    |   global total_dis = wv_total_hz * wave_dis
    | 
    |   # robot speed distance/time = speed
    |   wv_system_speed = total_dis / (wv_times)
    |   if(wv_times == 0 or cir_speed_org == 0):
    |     write_port_register(142,111)
    |     sleep(0.5)
    |     halt
    |   end
    |   return wv_system_speed
    | end
    | 
    | 
    | def set_current_voltage(o_cur,o_vol):
    |   if(isHicomm):
    |     set_current_voltage_hicomm(o_cur,o_vol)
    |   else:
    |     set_current_voltage_analog(o_cur,o_vol)
    |   end
    | end
    | 
    | def set_current_voltage_hicomm(o_cur,o_vol):
    |     write_port_register(204,o_cur)
    |     write_port_register(205,o_vol*10)
    |     write_port_register(133,o_cur)
    |     write_port_register(134,o_vol*10)
    | end
    | 
    | def set_current_voltage_analog(o_cur,o_vol):
    |     vol_an=((o_vol-14)/2.8)/10
    |     amp_an=((o_cur-60)/44)/10
    |     set_standard_analog_out(0,vol_an)
    |     set_standard_analog_out(1,amp_an)
    |     write_port_register(133,o_cur)
    |     write_port_register(134,o_vol*10)
    | end
    | 
    | def calculate_2f(wving_amplitude,tg_wv_wp1,tg_wv_wp2,cir_speed_org,wving_frequency,wving_delay,wving_crater,wving_dir):
    |   # 진폭
    |   global y_radius = wving_amplitude / 2
    |   # 이동 거리
    |   global move_dis = point_dist(tg_wv_wp1,tg_wv_wp2)*1000
    |   global move_dis_total = move_dis
    |   # total running time (sec) - cir_speed_org cpm.
    |   global wv_times_org = move_dis/(cir_speed_org/6)
    |   global wv_times = wv_times_org
    |   global wv_total_hz = floor(wv_times_org*wving_frequency/(1+wving_delay[0]+wving_delay[1]+wving_delay[2]+wving_delay[3]))
    |   global get_total = wv_total_hz
    | 
    |   dir=1
    | 
    |   ratio_t_sam = 1/get_total
    |   T1_sam = interpolate_pose(tg_wv_wp1,tg_wv_wp2,ratio_t_sam)
    |   ratio_t_sam = ratio_t_sam + 1/get_total
    |   T2_sam = interpolate_pose(tg_wv_wp1,tg_wv_wp2,ratio_t_sam)
    |   ratio_t_sam = ratio_t_sam + 1/get_total
    |   T3_sam = interpolate_pose(tg_wv_wp1,tg_wv_wp2,ratio_t_sam)
    | 
    |   push_angle = wving_crater[6]
    |   push_dis_sam = norm(y_radius)/tan(d2r(push_angle))
    |   Tp1_sam = feature_offset(T2_sam,p[0,y_radius/1000,0,0,0,0],wv_Line_Feature2)
    |   Tp2_sam = feature_offset(T2_sam,p[0,-y_radius/1000,0,0,0,0],wv_Line_Feature2)
    |   Tp1_sam = feature_offset(Tp1_sam,p[wving_dir*push_dis_sam/1000,0,0,0,0,0],wv_Line_Feature2)
    |   Tp3_sam = feature_offset(T3_sam,p[0,-y_radius/1000,0,0,0,0],wv_Line_Feature2)
    |   total_step = (get_line_dist(Tp1_sam,Tp2_sam)+get_line_dist(Tp1_sam,Tp3_sam))*1000
    |   total_dis = wv_total_hz * total_step
    | 
    |   wv_system_speed = (total_dis / wv_times)
    | 
    |   if(wv_times == 0 or cir_speed_org == 0):
    |     write_port_register(142,111)
    |     sleep(0.5)
    |     halt
    |   end
    |   return wv_system_speed
    | end
    | def weaving_simple(wv_wp1,wv_wp3,cir_speed_org,wving_frequency,wving_amplitude,welding_on):
    |   wv_dist = 0
    |   tilt_deg = [0,0,0]
    |   wving_delay = [0,0,0,0]
    |   wving_type = 1
    |   Arc_sen=[0,0,0,0,0,0]
    |   wv_gap=[0,0,0,0]
    |   welding_dir=1
    |   z_param=[0,0,0,0,0]
    |   par_2f=False
    |   wving_crater=[0,0,0,0,0,0,0,0,0,0]
    |   ext_fun=[0,0,0,0,0,0,0,0,0,0,0]
    |   wv_seq = [0,-1]
    |   wv_feature=p[0,0,0,0,0,0]
    |   wv_weldpar=[0,cir_speed_org,0,wving_frequency,wving_amplitude,wving_type,welding_dir]
    |   line_weaving_tp(wv_wp1,wv_wp3,wv_weldpar,tilt_deg,wving_delay,welding_on,Arc_sen,wv_gap,z_param,par_2f,wving_crater,ext_fun,wv_seq,wv_feature)
    | end
    | 
    | def line_weaving_tp(wv_wp1,wv_wp3,wv_weldpar=[100,10,0,1,5,1,1,1,0],tilt_deg=[0,0,0],wving_delay=[0,0,0,0],welding_on=False,Arc_sen=[0,0,0,0,0,0],wv_gap=[0,0,0,0],z_param=[0,0,0,0,0],par_2f=False,wving_crater=[0,0,0,0,0,0,0,0,0,0],ext_fun=[0,0,0,0,0,0,0,0,0,0,0],wv_seq = [0,-1],wv_feature=p[0,0,0,0,0,0]):
    |   global start_gas_time = 2
    |   global counter_average = 1
    |   global counter_average_num = 0
    |   global waste_cycle = ext_fun[8]
    |   if(first_half):
    |     Arc_sen[1] = Arc_sen[1]/2
    |     Arc_sen[2] = Arc_sen[2]/2
    |     Arc_sen[3] = Arc_sen[3]/2
    |     Arc_sen[4] = Arc_sen[4]/2
    |   end
    |   global arc_x_off=0
    |   global arc_z_off=0
    |   global Up = 0
    |   global Ui = 0
    |   global Up_z = 0
    |   global Ui_z = 0
    |   if(wv_weldpar[7] == 1):
    |     global record_multi = False
    |   else:
    |     global record_multi = True
    |   end
    |   global th_ext_fun = ext_fun
    |   RTDE_init()
    | 
    |   # e-Series 2, CB-Seris 8
    |   global system_bus_ms = 2
    | 
    |   global sin_dir = wv_seq[1]
    |   global start_trig = False
    |   dir=1
    |   if(par_2f):
    |     global squash_cycle = 0
    |     # sin_dir = sin_dir
    |     sin_dir = sin_dir * -1
    |   else:
    |     global squash_cycle = ext_fun[7]
    |   end
    |   global tri_count=0
    | 
    |   global z_bottom = z_param[0]/1000
    |   if(wv_weldpar[6]==-1):
    |     #right
    |     global vir_v = -1
    |   else:
    |     #left
    |     global vir_v = 1
    |   end
    | 
    |   if(par_2f):
    |     global cal_off_ang_rx = 1
    |     global cal_off_ang_ry = 0
    |   else:
    |     global cal_off_ang_rx = 0
    |     global cal_off_ang_ry = 1
    |   end
    | 
    |   if(wv_seq[0] == 2 or wv_seq[0] == 3):
    |     tilt_deg = [0,0,0]
    |     global cal_off_ang_rx = 0
    |     global cal_off_ang_ry = 0
    |   end
    | 
    |   global wv_Line_Feature2 = wv_wp1
    |   if(wv_weldpar[0] > 650 and par_2f == False):
    |     wv_weldpar[0] = 650
    |   end
    |   if(wv_wp3==p[0,0,0,0,0,0]):
    |     global wv_wp2 = feature_offset(wv_wp1,p[wv_weldpar[0]/1000,0,0,0,0,0],wv_Line_Feature2)
    |   else:
    |     global wv_wp2 = wv_wp3
    |     wv_weldpar[0] = point_dist(wv_wp1,wv_wp2)*1000
    |     global wv_dist_bak = point_dist(wv_wp1,wv_wp2)*1000
    |   end
    |   if(wv_feature != p[0,0,0,0,0,0]):
    |     wv_Line_Feature2 = wv_feature
    |   end
    |   if(vir_v==1):
    |     line_x = get_feature_Line(wv_wp1,wv_wp2)
    |   else:
    |     line_x = get_feature_Line(wv_wp2,wv_wp1)
    |   end
    |   pp1 = feature_offset(wv_wp1,p[0,20/1000,0,0,0,0],line_x)
    |   pp2 = pose_add(wv_wp1,p[0,0,20/1000,0,0,0])
    |   global wp_Feature = get_feature_plane_yz(wv_wp1,pp1,pp2)
    | 
    |   #setting
    |   if(par_2f):
    |     #todo - 1
    |     global offset_2f_k = -1 * ext_fun[9]
    |     global offset_2f_z = 1 * ext_fun[10]
    |     if(wv_seq[0] == 0 or wv_seq[0] == 1):
    |       # line_feature = get_feature_Line(wv_wp1,wv_wp2)
    |       line_feature = get_feature_Line(wv_wp2,wv_wp1)
    |       b_p1 = wv_wp1
    |       b_p2 = feature_offset(wv_wp1,p[0,0.02*vir_v,0,0,0,0],line_feature)
    |       # b_p2 = feature_offset(wv_wp1,p[0,0.01,0,0,0,0],line_feature)
    |       b_p3 = pose_add(wv_wp1,p[0,0,0.02,0,0,0])
    | 
    |       global back_feature = get_feature_plane_xz(b_p1,b_p2,b_p3)
    | 
    |       wv_wp1 = pose_trans(wv_wp1,p[0,0,0,0,0,d2r(-90)])
    |       wv_wp1 = feature_offset(wv_wp1,p[0,offset_2f_k/1000,0,0,0,0],back_feature)
    |       wv_wp1 = pose_add(wv_wp1,p[0,0,offset_2f_z/1000,0,0,0])
    |       global bak_wv_wp1 = wv_wp1
    |     end
    |       wv_wp2 = feature_offset(wv_wp2,p[0,offset_2f_k/1000,0,0,0,0],back_feature)
    |       wv_wp2 = pose_add(wv_wp2,p[0,0,offset_2f_z/1000,0,0,0])
    |       wv_wp2 = p[wv_wp2[0],wv_wp2[1],wv_wp2[2],wv_wp1[3],wv_wp1[4],wv_wp1[5]]
    |       global bak_wv_wp2 = wv_wp2
    |   end
    |   if(ext_fun[2]==1 and par_2f==False):
    |     w_voltage = ext_fun[3]
    |     w_current = ext_fun[4]
    |     set_current_voltage(w_current,w_voltage)
    |     global cir_speed_org_bak = wv_weldpar[1]
    |     global wving_amplitude_bak = wv_weldpar[4]
    |     wv_weldpar[1] = ext_fun[6]
    |     wv_weldpar[4] = ext_fun[5]
    |   end
    |   if(par_2f):
    |     global wv_system_speed = calculate_2f(wv_weldpar[4],wv_wp1,wv_wp2,wv_weldpar[1],wv_weldpar[3],wving_delay,wving_crater,wv_weldpar[6])
    |   else:
    |     global wv_system_speed = calculate_3f(wv_weldpar[4],wv_wp1,wv_wp2,wv_weldpar[1],wv_weldpar[3],wving_delay)
    |     x_radius = x_radius / 1000
    |   end
    |   global wv_set_speed = wv_system_speed
    |   ratio_t=0
    |   global y_radius = y_radius / 1000
    |   global y_radius_bak = y_radius
    |   global ext_stick = 0
    |   global th_arc_sen=Arc_sen
    |   global th_wv_gap=wv_gap
    |   global th_tilt_deg=tilt_deg
    |   global last_tilt_deg = th_tilt_deg
    |   global last_wv_wp1 = wv_wp1
    |   global last_wv_line = wv_Line_Feature2
    |   global last_z_bottom = z_bottom
    |   global th_wving_crater=wving_crater
    |   global th_par_2f = par_2f
    |   global th_cir_speed_org=wv_weldpar[1]
    |   global th_wv_wp1 = wv_wp1
    |   global th_wv_wp2 = wv_wp2
    |   global th_wv_wp3 = wv_wp3
    |   global th_wv_weldpar=wv_weldpar
    |   global th_wving_delay=wving_delay
    |   global th_z_param=z_param
    |   global th_wv_seq = wv_seq
    |   global th_wv_feature=wv_feature
    |   global th_dir = dir
    | 
    |   # if want to use approach position
    |   if(wv_seq[0] ==0 or wv_seq[0] == 1):
    |     global get_angle_rx = welding_angle_cal_2f(wv_wp1[1],tilt_deg,vir_v,cal_off_ang_rx)
    |     global get_angle_ry = welding_angle_cal_3f(wv_wp1[2],tilt_deg,z_bottom,cal_off_ang_ry)
    | 
    |     target_p = feature_offset(wv_wp1,p[0,0,0,d2r(tilt_deg[0] + get_angle_rx),d2r(tilt_deg[1] + get_angle_ry),d2r(tilt_deg[2])],wv_Line_Feature2)
    | 
    |     if(wv_weldpar[2]==1):
    |       target_p_appr = feature_offset(target_p,p[0,0,-0.02,0,0,0],wv_Line_Feature2)
    |       movel(target_p_appr,a=0.5,v=0.125)
    |     end
    |     movel(target_p,a=0.5,v=0.125)
    |   end
    |   CThread = run CalThread()
    |   DThread = run diff_Thread()
    |   TThread = run thread_timer()
    |   AThread = run Arc_Thread()
    |   TTRRhread = run thread_dist_rec()
    | 
    |   global timer_counting=True
    |   global program_weld_on = True
    | 
    |   if(a9_wv_weldingon==True):
    |     while(welding_off_t==55):
    |       sync()
    |     end
    |     if(wving_crater[2]>0):
    |       set_current_voltage(wving_crater[0],wving_crater[1])
    |     end
    |     if(welding_off_t != 1):
    |       if(isHicomm):
    |         write_welder(0,True)
    |       else:
    |         set_standard_digital_out(0,True)
    |       end
    |       while(read_welder(5)==False):
    |         if(weld_onoff==False):
    |             write_welder(0,True)
    |         end
    |         sync()
    |       end
    |       if(wving_crater[2]>0):
    |         #Crater Begin option
    |         write_output_float_register(1,1)
    |         sleep(wving_crater[2])
    |         set_current_voltage(ext_fun[1],ext_fun[0])
    |       end
    |     end
    |   end
    |   start_gas_time = 0
    | 
    |   background_cal=1
    |   background_ready=0
    |   FT_trig=True
    |   timer_1_is_counting = True
    |   global welding_program = False
    | 
    |   while((ratio_t < 1)):
    |     if( (norm(tri_count)>=2 and par_2f==False or FT_trig==True) or (norm(tri_count)>=4 and par_2f or FT_trig==True) ):
    |       FT_trig = False
    |       while(background_ready==0):
    |         sync()
    |       end
    |       tri_count = 0
    |       background_ready = 0
    |       global move_p = background_pose
    |       wv_wp2 = th_wv_wp2
    |       if(par_2f):
    |         background_cal=1
    |       else:
    |         background_cal=1
    |       end
    |       global a_val = 3
    |       if(a_val >= 30):
    |         write_port_register(142,112)
    |         sleep(0.5)
    |         halt
    |       end
    |     end
    |     if(wv_weldpar[5] ==1):
    |         if( (sin_dir==1 and wving_delay[0]==0) or (sin_dir==-1 and wving_delay[2]==0)):
    |          tri_count = tri_count + 1
    |         end
    |         global target_p = move_p[tri_count]
    |         # write_output_float_register(24,tri_count)
    |         # target_p=p[target_p[0],target_p[1],target_p[2],target_p[3],target_p[4],target_p[5]]
    |         tri_count = tri_count + 1
    |     elif(wv_weldpar[5] ==2):
    |       if((tri_count==0 and wving_delay[2]==0) or (tri_count==2 and wving_delay[0]==0)):
    |        tri_count = tri_count + 1
    |       end
    |       global target_p = move_p[tri_count]
    |       # write_output_float_register(24,tri_count)
    |       # target_p=p[target_p[0],target_p[1],target_p[2],target_p[3],target_p[4],target_p[5]]
    |       tri_count = tri_count + 1
    |     else:
    |       popup("Please insert 0 - sin or 1 - triangle")
    |     end
    |     if(target_p == p[0,0,0,0,0,0]):
    |       target_p = get_actual_tcp_pose()
    |     end
    |     #3F tri_count 2 는 tri_count가 계속 move_p[1]만 간다
    | 
    |     # write_output_float_register(23,sin_dir)
    | 
    |     ARC_T_ONOFF = True
    |     ARC_T_s_pose = get_actual_tcp_pose()
    |     ARC_T_e_pose = target_p
    |     if((norm(tri_count)== 2) and wving_delay[1]>0 and par_2f):
    |       #down
    |       movel(target_p,a=a_val,v=wv_system_speed/1000)
    |       sleep(wving_delay[1])
    |     elif((norm(tri_count)== 4) and wving_delay[3]>0 and par_2f):
    |       #4
    |       movel(target_p,a=a_val,v=wv_system_speed/1000)
    |       sleep(wving_delay[3])
    |     elif((norm(tri_count)== 2) and sin_dir==1 and wving_delay[1]>0 and par_2f == False):
    |       movel(target_p,a=a_val,v=wv_system_speed/1000)
    |       sleep(wving_delay[1])
    |     elif((norm(tri_count)== 2) and sin_dir==-1 and wving_delay[3]>0 and par_2f == False):
    |       movel(target_p,a=a_val,v=wv_system_speed/1000)
    |       sleep(wving_delay[3])
    |     elif((norm(tri_count)== 1) and wving_delay[2]>0 and par_2f):
    |       movel(target_p,a=a_val,v=wv_system_speed/1000)
    |       sleep(wving_delay[2])
    |     elif((norm(tri_count)== 3) and wving_delay[0]>0 and par_2f):
    |       #3
    |       movel(target_p,a=a_val,v=wv_system_speed/1000)
    |       sleep(wving_delay[0])
    |     else:
    |       movel(target_p,a=a_val,v=wv_system_speed/1000)
    |     end
    |     global last_pose = target_p
    |   end
    |   timer_1_is_counting = False
    | 
    |   if(a9_wv_weldingon == True and wving_crater[5]!=0):
    |     #crater end option
    |     set_current_voltage(wving_crater[3],wving_crater[4])
    |     sleep(wving_crater[5])
    |     program_weld_on = False
    |     set_current_voltage(ext_fun[1],ext_fun[0])
    |     if(isHicomm):
    |       write_port_register(202,0)
    |       write_port_register(149,0)
    |     else:
    |       set_standard_digital_out(0,False)
    |     end
    |     while(read_welder(5)==True):
    |       if(weld_onoff==True):
    |         write_welder(0,False)
    |       end
    |       sync()
    |     end
    |   end
    |   timer_counter = 0
    |   kill CThread
    |   kill DThread
    |   kill TThread
    |   kill AThread
    |   kill TTRRhread
    |   ARC_T_ONOFF=False
    |   timer_counter = 0
    |   timer_counting = False
    |   wcr_counter = 0
    |   wcr_counting = False
    |   get_wcr = False
    |   welding_off_t = 0
    |   plus_alpha_x = 0
    |   plus_alpha_z = 0
    | 
    |   if(wv_seq[0] == 0 or wv_seq[0] == 3):
    |     if(a9_wv_weldingon==True):
    |       program_weld_on = False
    |       write_port_register(202,0)
    |       write_port_register(149,0)
    |       write_welder(0,False)
    |       if(wv_weldpar[2]==1):
    |         target_pos = feature_offset(get_actual_tcp_pose(),p[0,0,-0.01,0,0,0],wv_Line_Feature2)
    |         movel(target_pos,0.5,0.01)
    |       end
    |     end
    |   end
    |   background_pose = [dumy_p,dumy_p,dumy_p,dumy_p]
    |   move_p = background_pose
    |   return sin_dir
    | end
    | 
    | 
    | def line_weaving_tp_l(wv_wp1,wv_wp3,wv_weldpar=[100,10,0,1,5,1,1,1,0],tilt_deg=[0,0,0],wving_delay=[0,0,0,0],welding_on=False,Arc_sen=[0,0,0,0,0,0],wv_gap=[0,0,0,0],z_param=[0,0,0,0,0],par_2f=False,wving_crater=[0,0,0,0,0,0,0,0,0,0],ext_fun=[0,0,0,0,0,0,0,0,0,0,0],wv_seq = [0,-1],wv_feature=p[0,0,0,0,0,0]):
    |   global start_gas_time = 2
    |   global counter_average = 1
    |   global counter_average_num = 0
    |   global waste_cycle = ext_fun[8]
    |   if(first_half):
    |     Arc_sen[1] = Arc_sen[1]/2
    |     Arc_sen[2] = Arc_sen[2]/2
    |     Arc_sen[3] = Arc_sen[3]/2
    |     Arc_sen[4] = Arc_sen[4]/2
    |   end
    |   global current_list = 0
    |   global wv_wp4 = wv_wp3
    |   global A_T1 = wv_wp4[0]
    |   global A_T2 = wv_wp4[1]
    |   global A_T3 = wv_wp4[2]
    | 
    |   global arc_x_off=0
    |   global arc_z_off=0
    |   global Up = 0
    |   global Ui = 0
    |   global Up_z = 0
    |   global Ui_z = 0
    |   global th_ext_fun = ext_fun
    |   if(wv_weldpar[7] == 1):
    |     global record_multi = False
    |   else:
    |     global record_multi = True
    |   end
    |   RTDE_init()
    | 
    |   if (wv_gap[0]==1):
    |     gap_check = True
    |     wv_gap[0]=0
    |   else:
    |     gap_check= False
    |   end
    |   # e-Series 2, CB-Seris 8
    |   global system_bus_ms = 2
    | 
    |   global sin_dir = wv_seq[1]
    |   if(par_2f):
    |     global squash_cycle = 0
    |     # sin_dir = sin_dir
    |     sin_dir = sin_dir * -1
    |   else:
    |     global squash_cycle = ext_fun[7]
    |   end
    |   global start_trig = False
    |   dir=1
    | 
    |   global tri_count=0
    | 
    |   global z_bottom = z_param[0]/1000
    |   if(wv_weldpar[6]==-1):
    |     global vir_v = -1
    |   else:
    |     global vir_v = 1
    |   end
    | 
    |   if(par_2f):
    |     global cal_off_ang_rx = 1
    |     global cal_off_ang_ry = 0
    |   else:
    |     global cal_off_ang_rx = 0
    |     global cal_off_ang_ry = 1
    |   end
    | 
    |   if(wv_seq[0] == 2 or wv_seq[0] == 3):
    |     tilt_deg = [0,0,0]
    |     global cal_off_ang_rx = 0
    |     global cal_off_ang_ry = 0
    |   end
    | 
    |   global wv_Line_Feature2 = wv_wp1
    |   if(wv_weldpar[0] > 700 and par_2f == False):
    |     wv_weldpar[0] = 700
    |   end
    |   if(wv_wp3[0]==p[0,0,0,0,0,0]):
    |     global wv_wp2 = feature_offset(wv_wp1,p[wv_weldpar[0]/1000,0,0,0,0,0],wv_Line_Feature2)
    |   else:
    |     global wv_wp2 = wv_wp4[0]
    |     wv_weldpar[0] = point_dist(wv_wp1,wv_wp2)*1000
    |     global wv_dist_bak = point_dist(wv_wp1,wv_wp2)*1000
    |   end
    |   if(wv_seq[0] == 2 or wv_seq[0] == 3):
    |     wv_Line_Feature2 = wv_feature
    |   end
    |   if(vir_v==1):
    |     line_x = get_feature_Line(wv_wp1,wv_wp2)
    |   else:
    |     line_x = get_feature_Line(wv_wp2,wv_wp1)
    |   end  pp1 = feature_offset(wv_wp1,p[0,20/1000,0,0,0,0],line_x)
    |   pp2 = pose_add(wv_wp1,p[0,0,20/1000,0,0,0])
    |   global wp_Feature = get_feature_plane_yz(wv_wp1,pp1,pp2)
    | 
    |   #setting
    |   if(par_2f):
    |     #todo - 1
    |     offset_2f_k = -1 * ext_fun[9]
    |     offset_2f_z = 1 * ext_fun[10]
    |     if(wv_seq[0] == 0 or wv_seq[0] == 1):
    |       line_feature = get_feature_Line(wv_wp1,wv_wp2)
    |       b_p1 = wv_wp1
    |       b_p2 = feature_offset(wv_wp1,p[0,0.01*vir_v,0,0,0,0],line_feature)
    |       b_p3 = pose_add(wv_wp1,p[0,0,0.01,0,0,0])
    | 
    |       back_feature = get_feature_plane_xz(b_p1,b_p2,b_p3)
    |       wv_wp1 = pose_trans(wv_wp1,p[0,0,0,0,0,d2r(-90)])
    |       wv_wp1 = feature_offset(wv_wp1,p[0,offset_2f_k/1000,0,0,0,0],back_feature)
    |       wv_wp1 = pose_add(wv_wp1,p[0,0,offset_2f_z/1000,0,0,0])
    |       # wv_wp1 = pose_add(wv_wp1,p[offset_2f_k/1000,0,0,0,0,0])
    |     end
    |       # wv_wp2 = pose_add(wv_wp2,p[offset_2f_k/1000,0,0,0,0,0])
    |       wv_wp2 = feature_offset(wv_wp2,p[0,offset_2f_k/1000,0,0,0,0],back_feature)
    |       wv_wp2 = pose_add(wv_wp2,p[0,0,offset_2f_z/1000,0,0,0])
    |       wv_wp2 = p[wv_wp2[0],wv_wp2[1],wv_wp2[2],wv_wp1[3],wv_wp1[4],wv_wp1[5]]
    | 
    |       wv_wp3_p = feature_offset(wv_wp3[0],p[0,offset_2f_k/1000,0,0,0,0],back_feature)
    |       wv_wp3_p = pose_add(wv_wp3_p,p[0,0,offset_2f_z/1000,0,0,0])
    |       wv_wp3_p = p[wv_wp3_p[0],wv_wp3_p[1],wv_wp3_p[2],wv_wp1[3],wv_wp1[4],wv_wp1[5]]
    |       wv_wp4[0] = p[wv_wp3_p[0],wv_wp3_p[1],wv_wp3_p[2],wv_wp1[3],wv_wp1[4],wv_wp1[5]]
    | 
    |       wv_wp3_p = feature_offset(wv_wp3[1],p[0,offset_2f_k/1000,0,0,0,0],back_feature)
    |       wv_wp3_p = pose_add(wv_wp3_p,p[0,0,offset_2f_z/1000,0,0,0])
    |       wv_wp3_p = p[wv_wp3_p[0],wv_wp3_p[1],wv_wp3_p[2],wv_wp1[3],wv_wp1[4],wv_wp1[5]]
    |       wv_wp4[1] = p[wv_wp3_p[0],wv_wp3_p[1],wv_wp3_p[2],wv_wp1[3],wv_wp1[4],wv_wp1[5]]
    | 
    |       wv_wp3_p = feature_offset(wv_wp3[2],p[0,offset_2f_k/1000,0,0,0,0],back_feature)
    |       wv_wp3_p = pose_add(wv_wp3_p,p[0,0,offset_2f_z/1000,0,0,0])
    |       wv_wp3_p = p[wv_wp3_p[0],wv_wp3_p[1],wv_wp3_p[2],wv_wp1[3],wv_wp1[4],wv_wp1[5]]
    |       wv_wp4[2] = p[wv_wp3_p[0],wv_wp3_p[1],wv_wp3_p[2],wv_wp1[3],wv_wp1[4],wv_wp1[5]]
    |   end
    |   if(ext_fun[2]==1 and par_2f==False):
    |     #squash
    |     w_voltage = ext_fun[3]
    |     w_current = ext_fun[4]
    |     set_current_voltage(w_current,w_voltage)
    |     global cir_speed_org_bak = wv_weldpar[1]
    |     global wving_amplitude_bak = wv_weldpar[4]
    |     wv_weldpar[1] = ext_fun[6]
    |     wv_weldpar[4] = ext_fun[5]
    |   end
    |   if(par_2f):
    |     global wv_system_speed = calculate_2f(wv_weldpar[4],wv_wp1,wv_wp2,wv_weldpar[1],wv_weldpar[3],wving_delay,wving_crater,wv_weldpar[6])
    |   else:
    |     global wv_system_speed = calculate_3f(wv_weldpar[4],wv_wp1,wv_wp2,wv_weldpar[1],wv_weldpar[3],wving_delay)
    |     x_radius = x_radius / 1000
    |   end
    |   global wv_set_speed = wv_system_speed
    |   ratio_t=0
    |   # mm -> m
    |   global y_radius = y_radius / 1000
    |   global y_radius_bak = y_radius
    |   #init for thread
    |   global ext_stick = 0
    |   global th_arc_sen=Arc_sen
    |   global th_wv_gap=wv_gap
    |   global th_tilt_deg=tilt_deg
    | 
    |   global last_tilt_deg =th_tilt_deg
    |   global last_wv_wp1 = wv_wp1
    |   global last_wv_line = wv_Line_Feature2
    |   global th_wving_crater=wving_crater
    |   global last_z_bottom = z_bottom
    |   global th_par_2f = par_2f
    |   global th_cir_speed_org=wv_weldpar[1]
    |   global th_wv_wp1 = wv_wp1
    |   global th_wv_wp2 = wv_wp2
    |   global th_wv_wp3 = wv_wp3[0]
    |   global th_wv_weldpar=wv_weldpar
    |   global th_wving_delay=wving_delay
    |   global th_z_param=z_param
    |   global th_wv_seq = wv_seq
    |   global th_wv_feature=wv_feature
    |   global th_dir = dir
    | 
    |   # if want to use approach position
    |   if(wv_seq[0] ==0 or wv_seq[0] == 1):
    |     global get_angle_rx = welding_angle_cal_2f(wv_wp1[1],tilt_deg,vir_v,cal_off_ang_rx)
    |     global get_angle_ry = welding_angle_cal_3f(wv_wp1[2],tilt_deg,z_bottom,cal_off_ang_ry)
    | 
    |     target_p = feature_offset(wv_wp1,p[0,0,0,d2r(tilt_deg[0] + get_angle_rx),d2r(tilt_deg[1] + get_angle_ry),d2r(tilt_deg[2])],wv_Line_Feature2)
    | 
    |     if(wv_weldpar[2]==1):
    |       target_p_appr = feature_offset(target_p,p[0,0,-0.02,0,0,0],wv_Line_Feature2)
    |       movel(target_p_appr,a=0.5,v=0.125)
    |     end
    |     movel(target_p,a=0.5,v=0.125)
    |   end
    | 
    |   CThread = run CalThread()
    |   DThread = run diff_Thread()
    |   TThread = run thread_timer()
    |   AThread = run Arc_Thread()
    |   TTRRhread = run thread_dist_rec()
    | 
    |   global timer_counting=True
    |   global program_weld_on = True
    | 
    |   if(a9_wv_weldingon==True):
    |     while(welding_off_t==55):
    |       sync()
    |     end
    |     if(wving_crater[2]>0):
    |       set_current_voltage(wving_crater[0],wving_crater[1])
    |     end
    |     if(welding_off_t != 1):
    |       write_welder(0,True)
    |       while(get_wcr==False):
    |         if(weld_onoff==False):
    |           write_welder(0,True)
    |         end
    |         sync()
    |       end
    |       if(wving_crater[2]>0):
    |         #Crater Begin option
    |         write_output_float_register(1,1)
    |         sleep(wving_crater[2])
    |         set_current_voltage(ext_fun[1],ext_fun[0])
    |       end
    |     end
    |   end
    |   start_gas_time = 0
    | 
    |   background_cal=1
    |   background_ready=0
    |   FT_trig=True
    | 
    |   timer_1_is_counting = True
    | 
    |   while((ratio_t < 1) or current_list==0 or current_list==1):
    |     if(ratio_t>=1 and current_list!=2):
    |       if (gap_check):
    |         gap_check = True
    |         wv_gap[0]=1
    |         th_wv_gap[0]=1
    |         gap_check= False
    |       end
    |       ratio_t=0
    |       if(current_list==0):
    |         wving_amp_bak = wv_weldpar[4]
    |         wv_weldpar[4] = wv_weldpar[4] * 1
    |         th_wv_weldpar[4] = wv_weldpar[4]
    |         circle_speed_bak = wv_weldpar[1]
    |         wv_weldpar[1]= wv_weldpar[1]*0.7
    |         th_wv_weldpar[1]= wv_weldpar[1]
    |       elif(current_list==1):
    |         wv_weldpar[4] = wving_amp_bak
    |         th_wv_weldpar[4] = wv_weldpar[4]
    |         wv_weldpar[1] = circle_speed_bak
    |         th_wv_weldpar[1]= wv_weldpar[1]
    |       end
    |       wv_wp1=wv_wp4[current_list]
    |       wv_wp2=wv_wp4[current_list+1]
    |       global th_wv_wp1 = wv_wp4[current_list]
    |       global th_wv_wp2 = wv_wp4[current_list+1]
    |       global th_wv_wp3 = wv_wp4[current_list+1]
    |       wv_system_speed_bak = wv_system_speed
    |       if(par_2f):
    |         global wv_system_speed = calculate_2f(wv_weldpar[4],wv_wp4[current_list],wv_wp4[current_list+1],wv_weldpar[1],wv_weldpar[3],wving_delay,wving_crater)
    |         global y_radius = y_radius / 1000
    |         global y_radius_bak = y_radius
    |       else:
    |         global wv_system_speed = calculate_3f(wv_weldpar[4],wv_wp4[current_list],wv_wp4[current_list+1],wv_weldpar[1],wv_weldpar[3],wving_delay)
    |         x_radius = x_radius / 1000
    |       end
    |       wv_system_speed = wv_system_speed_bak
    |       current_list=current_list+1
    |     end
    | 
    |     if( (norm(tri_count)>=2 and par_2f==False or FT_trig==True) or (norm(tri_count)>=4 and par_2f==True or FT_trig==True)   ):
    |       FT_trig = False
    |       while(background_ready==0):
    |         sync()
    |       end
    |       tri_count = 0
    |       background_ready = 0
    |       global move_p = background_pose
    |       wv_wp2 = th_wv_wp2
    |       if(par_2f):
    |         background_cal=1
    |       else:
    |         background_cal=1
    |       end
    |       global a_val = 3
    |       if(a_val >= 30):
    |         write_port_register(142,112)
    |         sleep(0.5)
    |         halt
    |       end
    |     end
    | 
    |     if(wv_weldpar[5] ==1):
    |         if( (sin_dir==1 and wving_delay[0]==0) or (sin_dir==-1 and wving_delay[2]==0)):
    |          tri_count = tri_count + 1
    |         end
    |         # write_output_float_register(24,tri_count)
    |         global target_p = move_p[tri_count]
    |         target_p=p[target_p[0],target_p[1],target_p[2],target_p[3],target_p[4],target_p[5]]
    |         tri_count = tri_count + 1
    |     elif(wv_weldpar[5] ==2):
    |       if( (tri_count==1 and sin_dir==1 and wving_delay[0]==0) or (tri_count==1 and sin_dir==-1 and wving_delay[2]==0)):
    |        tri_count = tri_count + 1
    |       end
    |       # write_output_float_register(24,tri_count)
    |       global target_p = move_p[tri_count]
    |       target_p=p[target_p[0],target_p[1],target_p[2],target_p[3],target_p[4],target_p[5]]
    |       tri_count = tri_count + 1
    |     else:
    |       popup("Please insert 0 - sin or 1 - triangle")
    |     end
    | 
    |     if(target_p == p[0,0,0,0,0,0]):
    |       target_p = get_actual_tcp_pose()
    |     end
    |     # write_output_float_register(23,sin_dir)
    |     ARC_T_ONOFF = True
    |     ARC_T_s_pose = get_actual_tcp_pose()
    |     ARC_T_e_pose = target_p
    |     if((norm(tri_count)== 2) and wving_delay[1]>0 and par_2f):
    |       # DOWN
    |       movel(target_p,a=a_val,v=wv_system_speed/1000)
    |       sleep(wving_delay[1])
    |     elif((norm(tri_count)== 4) and wving_delay[3]>0 and par_2f):
    |       #UP
    |       movel(target_p,a=a_val,v=wv_system_speed/1000)
    |       sleep(wving_delay[3])
    |     elif((norm(tri_count)== 2) and sin_dir==1 and wving_delay[1]>0 and par_2f == False):
    |       movel(target_p,a=a_val,v=wv_system_speed/1000)
    |       sleep(wving_delay[1])
    |     elif((norm(tri_count)== 2) and sin_dir==-1 and wving_delay[3]>0 and par_2f == False):
    |       movel(target_p,a=a_val,v=wv_system_speed/1000)
    |       sleep(wving_delay[3])
    |     elif((norm(tri_count)== 1) and wving_delay[0]>0 and par_2f):
    |       movel(target_p,a=a_val,v=wv_system_speed/1000)
    |       sleep(wving_delay[0])
    |     elif((norm(tri_count)== 3) and wving_delay[2]>0 and par_2f):
    |       movel(target_p,a=a_val,v=wv_system_speed/1000)
    |       sleep(wving_delay[2])
    |     else:
    |       movel(target_p,a=a_val,v=wv_system_speed/1000)
    |     end
    |     global last_pose = target_p
    |   end
    | 
    |   timer_1_is_counting = False
    |   welding_program = True
    |   if(a9_wv_weldingon == True and wving_crater[5]!=0):
    |     #crater end option
    |     set_current_voltage(wving_crater[3],wving_crater[4])
    |     sleep(wving_crater[5])
    |     program_weld_on = False
    |     set_current_voltage(ext_fun[1],ext_fun[0])
    |     if(isHicomm):
    |       write_port_register(202,0)
    |       write_port_register(149,0)
    |     else:
    |       set_standard_digital_out(0,False)
    |     end
    |     while(get_wcr==True):
    |       if(weld_onoff==True):
    |         if(isHicomm):
    |           write_port_register(202,0)
    |           write_port_register(149,0)
    |         else:
    |           set_standard_digital_out(0,False)
    |         end
    |       end
    |       sync()
    |     end
    |   end
    | 
    |   kill CThread
    |   kill DThread
    |   kill TThread
    |   kill AThread
    |   kill TTRRhread
    |   ARC_T_ONOFF=False
    |   timer_counting = False
    |   wcr_counter = 0
    |   wcr_counting = False
    |   get_wcr = False
    |   welding_off_t = 0
    |   plus_alpha_x = 0
    |   plus_alpha_z = 0
    | 
    |   if(wv_seq[0] == 0 or wv_seq[0] == 3):
    |     if(a9_wv_weldingon==True):
    |       program_weld_on = False
    |       if(isHicomm):
    |         write_port_register(202,0)
    |         write_port_register(149,0)
    |       else:
    |         set_standard_digital_out(0,False)
    |       end
    |       if(wv_weldpar[2]==1):
    |         target_pos = feature_offset(get_actual_tcp_pose(),p[0,0,-0.01,0,0,0],wv_Line_Feature2)
    |         movel(target_pos,0.5,0.01)
    |       end
    |     end
    |   end
    |   background_pose = [dumy_p,dumy_p,dumy_p,dumy_p]
    |   move_p = background_pose
    |   return sin_dir
    | end
  Folder Reset [hidden by the author, left out]
  Folder Welding_Init [hidden by the author, left out]
  Folder init_reset_modbus_server [hidden by the author, left out]
Robot Program (runOnlyOnce=false)
  SuppressedNode
    Folder Folder [hidden by the author, left out]
  If simulation_mode
    'work mode 2'
    Script: write_port_register(162,2)
    touch_temp := 0
  If a0_Job_Mode≟1
    Folder job mode 1 [hidden by the author, left out]
    Call robotand_cell_initalizat
  ElseIf a0_Job_Mode≟2 (checkContinuously=true)
    'JOB_AUTO'
    auto_on := True
    Folder Init [hidden by the author, left out]
    Folder Cell_calculation [hidden by the author, left out]
    Auto_cur_cell := 0
    Folder Touch,Welding
      'Calculate total sequence and decide way'
      Folder Calculate & Move & Touch
        Folder touch_init [hidden by the author, left out]
        If touch_temp≟0
          Script: write_port_register(138,0)
          Call reset_multi_record
          Folder get_touch_position
            Folder get pre-positions
              If read_port_register(work_type_165)≟2
                Folder freedrive touch [hidden by the author, left out]
              Else 
                Folder value from pendant
                  move_i := 1
                  SuppressedNode
                    calcu_trig := True
                  Folder Touch_FrontandSide
                    If EXT_flag1[11]≟ True
                      Folder Touch front and side_Right [hidden by the author, left out]
                    Else 
                      Folder Touch front and side_Left [hidden by the author, left out]
                  SuppressedNode
                    Wait Condition expression=calcu_trig≟ False
                  Wait Condition expression=event_cal_on≟ False
                  SuppressedNode
                    Wait Condition expression=event_side_on≟ False
            Folder move and touch
              Folder Touch Move [hidden by the author, left out]
              Folder Touch After Offset [hidden by the author, left out]
              'Touch Remember On/OFF'
              Script: write_port_register(180,1)
        Else 
          Folder Ignore Touch and check error [hidden by the author, left out]
      Folder welding
        Folder weldings
          Auto_cur_cell := read_port_register(138)
          time_cal_trig := True
          Loop While (checkContinuously=false) expression=Auto_cur_cell<Auto_total_cell
            Script: write_port_register(138,Auto_cur_cell)
            running_trig := True
            '[2F_AB - 30] , [2F_CD_LEFT - 100] , [2F_CD_RIGHT - 150] , [3F - ELSE]'
            If Auto_W_num[Auto_cur_cell]≥100 and Auto_W_num[Auto_cur_cell]≤149
              '2F CD LEFT'
              A_sel_v := A_HOR
              A_sel_v_end := A_HOR_ML
              A_sel_v2 := A_HOR_M
              A_sel_v_end2 := A_HOR_R
              If floor(Auto_W_num[Auto_cur_cell]/10)≟10
                current_path := 1
                multi_path := 1
              ElseIf floor(Auto_W_num[Auto_cur_cell]/10)≟11
                current_path := 2
                multi_path := 2
              ElseIf floor(Auto_W_num[Auto_cur_cell]/10)≟12
                current_path := 3
                multi_path := 3
              ElseIf floor(Auto_W_num[Auto_cur_cell]/10)≟13
                current_path := 4
                multi_path := 4
              current_2f := current_2f+1
              CD_MLR := True
              Script: write_port_register(135,A_HOR)
              Script: write_port_register(136,current_2f)
              If simulation_mode
                Call welding_parameter_sim
              Else 
                Call welding_parameter_init
              wv_direction := 1
              If Auto_W_num[Auto_cur_cell]%10≟4
                A_sel_v := A_HOR_R
                Call MoveFun
                A_sel_v := A_HOR
              ElseIf Auto_W_num[Auto_cur_cell]%10≟0 or Auto_W_num[Auto_cur_cell]%10≟1 or Auto_W_num[Auto_cur_cell]%10≟2
                Call MoveFun
              Call weav_welding_2f_CD
            ElseIf Auto_W_num[Auto_cur_cell]≥150 and Auto_W_num[Auto_cur_cell]≤189
              '2F CD RIGHT'
              A_sel_v := A_HOR_R
              A_sel_v_end := A_HOR_MR
              A_sel_v2 := A_HOR_M
              A_sel_v_end2 := A_HOR
              If floor(Auto_W_num[Auto_cur_cell]/10)≟15
                current_path := 1
                multi_path := 1
              ElseIf floor(Auto_W_num[Auto_cur_cell]/10)≟16
                current_path := 2
                multi_path := 2
              ElseIf floor(Auto_W_num[Auto_cur_cell]/10)≟17
                current_path := 3
                multi_path := 3
              ElseIf floor(Auto_W_num[Auto_cur_cell]/10)≟18
                current_path := 4
                multi_path := 4
              current_2f := current_2f+1
              CD_MLR := False
              Script: write_port_register(135,A_HOR)
              Script: write_port_register(136,current_2f)
              If simulation_mode
                Call welding_parameter_sim
              Else 
                Call welding_parameter_init
              wv_direction := -1
              If Auto_W_num[Auto_cur_cell]%10≟4
                A_sel_v := A_HOR
                Call MoveFun
                A_sel_v := A_HOR_R
              ElseIf Auto_W_num[Auto_cur_cell]%10≟0 or Auto_W_num[Auto_cur_cell]%10≟1 or Auto_W_num[Auto_cur_cell]%10≟2
                Call MoveFun
              Call weav_welding_2f_CD
            ElseIf Auto_W_num[Auto_cur_cell]≥30 and Auto_W_num[Auto_cur_cell]≤65
              '2F'
              A_sel_v := A_HOR
              A_sel_v_end := A_HOR_R
              If floor(Auto_W_num[Auto_cur_cell]/10)≟3
                current_path := 1
                multi_path := 1
              ElseIf floor(Auto_W_num[Auto_cur_cell]/10)≟4
                current_path := 2
                multi_path := 2
              ElseIf floor(Auto_W_num[Auto_cur_cell]/10)≟5
                current_path := 3
                multi_path := 3
              ElseIf floor(Auto_W_num[Auto_cur_cell]/10)≟6
                current_path := 4
                multi_path := 4
              current_2f := current_2f+1
              Script: write_port_register(135,A_HOR)
              Script: write_port_register(136,current_2f)
              If simulation_mode
                Call welding_parameter_sim
              Else 
                Call welding_parameter_init
              If Auto_W_num[Auto_cur_cell]%10≟2
                A_sel_v := A_HOR_R
                Call MoveFun
                A_sel_v := A_HOR
              Else 
                Call MoveFun
              Call weav_welding_2f
            Else 
              A_sel_v := Auto_W_num[Auto_cur_cell]
              Script: write_port_register(135,A_sel_v)
              current_path := 1
              current_2f := 0
              Script: write_port_register(136,current_2f)
              If simulation_mode
                Call welding_parameter_sim
              Else 
                Call welding_parameter_init
              A_sel_v_end := A_sel_v+9
              Call weav_welding_3f
            Call reset_weld_param
            Folder next_before [hidden by the author, left out]
          Script: homeing()
          Script: write_port_register(162,1)
          Script: write_port_register(180,0)
  Wait Sleep waitTime=0.01
  Folder after init auto [hidden by the author, left out]
Thread Thread_2 (runOnlyOnce=false)
  Folder Thread_heartbeat [hidden by the author, left out]
Thread Thread_1 (runOnlyOnce=false)
  Folder thread main [hidden by the author, left out]
Event  expression=event_cal_on
  Folder calculate_position
    SuppressedNode
      A_Speed_list := [0, 0, 0, 0, 0, 0, 0, 0, 0, 0, 0, 0, 0, 0, 0, 0]
    SuppressedNode
      A_Distance_list := [0, 0, 0, 0, 0, 0, 0, 0, 0, 0, 0, 0, 0, 0, 0, 0]
    move_i_f := 1
    get_pose_side := 0
    Loop While (checkContinuously=false) expression=move_i_f<10
      If A_Touch_trig_l[move_i_f]≟ True
        If move_i_f≟A_VL1 or move_i_f≟A_VL2
          A_sel_v := move_i_f
          If simulation_mode
            Call welding_parameter_sim
          Else 
            Call welding_parameter_init
          If a8_wv_distance<5
            Script: write_port_register(142,143)
            Halt
          b2_left_par := True
          b8_wv_2f := False
          If move_i_f≟A_VL2
            callar_hor := a6_callar_hor
            If b1_cell_info_L≟E or b1_cell_info_L≟e
              'For bottom touch(zero) after offset not used now'
              vert_scallup_l := a5_f_hole[1]
            b2_cell := b1_cell_info_L
            get_pos := get_lr(up_left,a6_f_width,a5_f_hole,a7_f_distance,b2_left_par,b8_wv_2f,Touch_dis,get_margin_z,touch_side,callar_hor,b2_cell,center_line)
            SuppressedNode
              If b1_cell_info_L≟c or b1_cell_info_L≟d or b1_cell_info_L≟E or b1_cell_info_L≟e removedSiblings(If(type=Else checkContinuously=false, children(Assignment(valueSource=Expression, variable=b2_cell, expression=0))))
                b2_cell := b1_cell_info_L
          Else 
            callar_hor := 0
            'For bottom touch(zero) after offset not used now'
            vert_scallup_l := a5_f_hole[1]
            b2_cell := b1_cell_info_L
            get_pos := get_lr(left,a6_f_width,a5_f_hole,a7_f_distance,b2_left_par,b8_wv_2f,Touch_dis,get_margin_z,touch_side,callar_hor,b2_cell,center_line)
          pre_tp := tilt_3f_fun(get_pos,[0,0,0],0)
          Script: A_Prepos_l[move_i_f]=pre_tp
        ElseIf move_i_f≟A_VR1 or move_i_f≟A_VR2
          A_sel_v := move_i_f
          If simulation_mode
            Call welding_parameter_sim
          Else 
            Call welding_parameter_init
          If a8_wv_distance<5
            Script: write_port_register(142,143)
            Halt
          b2_left_par := False
          b8_wv_2f := False
          If move_i_f≟A_VR2
            callar_hor := a6_callar_hor
            If b1_cell_info_R≟E or b1_cell_info_R≟e
              vert_scallup_r := a5_f_hole[1]
            b2_cell := b1_cell_info_R
            get_pos := get_lr(up_right,a6_f_width,a5_f_hole,a7_f_distance,b2_left_par,b8_wv_2f,Touch_dis,get_margin_z,touch_side,callar_hor,b2_cell,center_line)
            SuppressedNode
              If b1_cell_info_R≟c or b1_cell_info_R≟d or b1_cell_info_R≟E or b1_cell_info_R≟e removedSiblings(If(type=Else checkContinuously=false, children(Assignment(valueSource=Expression, variable=b2_cell, expression=0))))
                b2_cell := b1_cell_info_R
          Else 
            callar_hor := 0
            vert_scallup_r := a5_f_hole[1]
            b2_cell := b1_cell_info_R
            get_pos := get_lr(right,a6_f_width,a5_f_hole,a7_f_distance,b2_left_par,b8_wv_2f,Touch_dis,get_margin_z,touch_side,callar_hor,b2_cell,center_line)
          pre_tp := tilt_3f_fun(get_pos,[0,0,0],0)
          Script: A_Prepos_l[move_i_f]=pre_tp
        ElseIf move_i_f≟A_HOR
          A_sel_v := A_HOR
          If simulation_mode
            Call welding_parameter_sim
          Else 
            Call welding_parameter_init
          hor_l_scallup := a5_f_hole[1]
          b8_wv_2f := True
          b2_left_par := True
          b2_cell := b1_cell_info_L
          get_pos := get_lr(up_left,a6_f_width,a5_f_hole,a7_f_distance,b2_left_par,b8_wv_2f,Touch_dis,get_margin_z,touch_side,0,b2_cell,center_line)
          pre_tp := get_pos
          Script: A_Prepos_l[move_i_f]=pre_tp
        ElseIf move_i_f≟A_HOR_R
          A_sel_v := A_HOR
          If simulation_mode
            Call welding_parameter_sim
          Else 
            Call welding_parameter_init
          hor_r_scallup := a5_f_hole[2]
          b2_left_par := False
          b8_wv_2f := True
          b2_cell := b1_cell_info_R
          get_pos := get_lr(up_right,a6_f_width,a5_f_hole,a7_f_distance,b2_left_par,b8_wv_2f,Touch_dis,get_margin_z,touch_side,0,b2_cell,center_line)
          pre_tp := get_pos
          Script: A_Prepos_l[move_i_f]=pre_tp
        ElseIf move_i_f≟A_HOR_ML
          A_sel_v := A_HOR_ML
          If simulation_mode
            Call welding_parameter_sim
          Else 
            Call welding_parameter_init
          b8_wv_2f := True
          b2_left_par := True
          b2_cell := b1_cell_info_L
          Touch_dis := -1*Touch_dis
          get_pos := get_lr(up_left,a6_f_width,a5_f_hole,a7_f_distance,b2_left_par,b8_wv_2f,Touch_dis,get_margin_z,touch_side,a6_callar_hor,b2_cell,center_line)
          Touch_dis := -1*Touch_dis
          pre_tp := get_pos
          Script: A_Prepos_l[move_i_f]=pre_tp
        ElseIf move_i_f≟A_HOR_MR
          A_sel_v := A_HOR_MR
          If simulation_mode
            Call welding_parameter_sim
          Else 
            Call welding_parameter_init
          b2_left_par := False
          b8_wv_2f := True
          b2_cell := b1_cell_info_R
          Touch_dis := -1*Touch_dis
          get_pos := get_lr(up_right,a6_f_width,a5_f_hole,a7_f_distance,b2_left_par,b8_wv_2f,Touch_dis,get_margin_z,touch_side,a6_callar_hor,b2_cell,center_line)
          Touch_dis := -1*Touch_dis
          pre_tp := get_pos
          Script: A_Prepos_l[move_i_f]=pre_tp
        If move_i_f≤4
          Script: A_Prepos_l[move_i_f+9]=p[0,0,0,0,0,0]
        SuppressedNode
          Script: A_Speed_list[move_i]=a2_speed_cpm
        SuppressedNode
          Script: A_Distance_list[move_i]=a8_wv_distance
      move_i_f := move_i_f+1
    event_cal_on := False
Event  expression=event_side_on
  Folder calculate_side [hidden by the author, left out]
Event  expression=reset_trig
  Call reset_weld_param
  reset_trig := False
Event  expression=time_cal_trig
  t_time := time_cal(Auto_W_num,Auto_total_cell,A_Speed_list,A_Distance_list,A_Touch_p,0)
  Script: write_port_register(144,t_time)
  time_cal_trig := False
Event  expression=pause_trig
  s_conn := socket_open("192.168.1.7",29999)
  s_send := socket_send_string("pause")
  s_send := socket_send_byte(10)
  Script: socket_close()
  pause_trig := False
SubProgram  [hidden by the author, left out]
SubProgram  [hidden by the author, left out]
SubProgram  [hidden by the author, left out]
SubProgram  [hidden by the author, left out]
SubProgram  [hidden by the author, left out]
SubProgram  [hidden by the author, left out]
SubProgram  [hidden by the author, left out]
SubProgram  [hidden by the author, left out]
SubProgram  [hidden by the author, left out]
SubProgram  [hidden by the author, left out]
SubProgram  [hidden by the author, left out]
SubProgram -> weav_welding_2f
SubProgram -> weav_welding_2f_CD
SubProgram  [hidden by the author, left out]
SubProgram  [hidden by the author, left out]
SubProgram reset_multi_record [hidden by the author, left out]
SubProgram weav_welding_2f_CD (keepSynchronizedWithDisk=false)
  If running_trig≟ True (checkContinuously=true)
    Folder CD_calculation [hidden by the author, left out]
    Folder gap_half [hidden by the author, left out]
    If EXT_flag1[4]≟ True  and (b1_cell_info_L≠c and b1_cell_info_L≠d and b1_cell_info_R≠c and b1_cell_info_R≠d)
      If EXT_flag1[6]
        If Auto_W_num[Auto_cur_cell]%10≟1
          Script: inv_inching(inv_inch_time)
          step_2f := 1
          Script: welding_result = line_weaving_tp_l(pos_m_path_cd,[pos_m_p_end_cd,pos_m_path,A_middle_weld],[a8_wv_distance,Circle_Speed,b1_appro_param,a4_wv_frequency,a3_wv_amplitude,b8_wv_type,wv_direction,current_path,c8_arc_cur_offs],b7_tilt_degree,b3_dealy_all,a9_wv_weldingon,c3_wv_arc,c7_wv_gap,a5_f_hole,b8_wv_2f,a7_weld_crater,squash_l)
        If Auto_W_num[Auto_cur_cell]%10≟4
          Script: inv_inching(inv_inch_time)
          a7_weld_crater := [d_start_current,d_start_voltage,d_start_time,d_end_current_2,d_end_voltage_2,d_end_time_2,d_lean_degree]
          Folder gap_half [hidden by the author, left out]
          step_2f := 2
          wv_direction := -1*wv_direction
          SuppressedNode
            A_middle_weld := feature_offset(A_middle_weld,p[20*wv_direction/1000,0,0,0,0,0],A_Touch_p[A_sel_v2])
          Script: welding_result = line_weaving_tp(pos_m_path_end,A_middle_weld,[a8_wv_distance,Circle_Speed,b1_appro_param,a4_wv_frequency,a3_wv_amplitude,b8_wv_type,wv_direction,current_path,c8_arc_cur_offs],b7_tilt_degree,b3_dealy_all,a9_wv_weldingon,c3_wv_arc,c7_wv_gap,a5_f_hole,b8_wv_2f,a7_weld_crater,squash_l)
      Else 
        If Auto_W_num[Auto_cur_cell]%10≟0
          Script: inv_inching(inv_inch_time)
          step_2f := 1
          Script: welding_result = line_weaving_tp_l(pos_m_path_cd,[pos_m_p_end_cd,pos_m_path,pos_m_path_end],[a8_wv_distance,Circle_Speed,b1_appro_param,a4_wv_frequency,a3_wv_amplitude,b8_wv_type,wv_direction,current_path,c8_arc_cur_offs],b7_tilt_degree,b3_dealy_all,a9_wv_weldingon,c3_wv_arc,c7_wv_gap,a5_f_hole,b8_wv_2f,a7_weld_crater,squash_l)
        Else 
          Script: write_port_register(142,142)
          Halt
    Else 
      If EXT_flag1[6]
        If Auto_W_num[Auto_cur_cell]%10≟2
          Script: inv_inching(inv_inch_time)
          step_2f := 1
          Folder gap_half [hidden by the author, left out]
          Script: welding_result = line_weaving_tp(pos_m_path_cd,pos_m_p_end_cd,[a8_wv_distance,Circle_Speed,b1_appro_param,a4_wv_frequency,a3_wv_amplitude,b8_wv_type,wv_direction,current_path,c8_arc_cur_offs],b7_tilt_degree,b3_dealy_all,a9_wv_weldingon,c3_wv_arc,c7_wv_gap,a5_f_hole,b8_wv_2f,a7_weld_crater,squash_l)
          Wait Sleep waitTime=0.5
        If Auto_W_num[Auto_cur_cell]%10≟3
          Script: inv_inching(inv_inch_time)
          step_2f := 2
          Script: welding_result = line_weaving_tp(pos_m_path,A_middle_weld,[a8_wv_distance,Circle_Speed,b1_appro_param,a4_wv_frequency,a3_wv_amplitude,b8_wv_type,wv_direction,current_path,c8_arc_cur_offs],b7_tilt_degree,b3_dealy_all,a9_wv_weldingon,c3_wv_arc,c7_wv_gap,a5_f_hole,b8_wv_2f,a7_weld_crater,squash_l)
          Wait Sleep waitTime=0.5
        If Auto_W_num[Auto_cur_cell]%10≟4
          Script: inv_inching(inv_inch_time)
          a7_weld_crater := [d_start_current,d_start_voltage,d_start_time,d_end_current_2,d_end_voltage_2,d_end_time_2,d_lean_degree]
          step_2f := 3
          Folder gap_half [hidden by the author, left out]
          wv_direction := -1*wv_direction
          SuppressedNode
            A_middle_weld := feature_offset(A_middle_weld,p[20*wv_direction/1000,0,0,0,0,0],A_Touch_p[A_sel_v2])
          Script: welding_result = line_weaving_tp(pos_m_path_end,A_middle_weld,[a8_wv_distance,Circle_Speed,b1_appro_param,a4_wv_frequency,a3_wv_amplitude,b8_wv_type,wv_direction,current_path,c8_arc_cur_offs],b7_tilt_degree,b3_dealy_all,a9_wv_weldingon,c3_wv_arc,c7_wv_gap,a5_f_hole,b8_wv_2f,a7_weld_crater,squash_l)
      Else 
        If Auto_W_num[Auto_cur_cell]%10≟2
          Script: inv_inching(inv_inch_time)
          step_2f := 1
          c7_wv_gap := [0,c5_wv_gap_y,c6_wv_gap_cpm,c9_wv_gap_freq]
          Script: welding_result = line_weaving_tp(pos_m_path_cd,pos_m_p_end_cd,[a8_wv_distance,Circle_Speed,b1_appro_param,a4_wv_frequency,a3_wv_amplitude,b8_wv_type,wv_direction,current_path,c8_arc_cur_offs],b7_tilt_degree,b3_dealy_all,a9_wv_weldingon,c3_wv_arc,c7_wv_gap,a5_f_hole,b8_wv_2f,a7_weld_crater,squash_l)
          Wait Sleep waitTime=0.5
        If Auto_W_num[Auto_cur_cell]%10≟5
          Script: inv_inching(inv_inch_time)
          step_2f := 2
          c7_wv_gap := [c4_gap_enable,c5_wv_gap_y,c6_wv_gap_cpm,c9_wv_gap_freq]
          Script: welding_result = line_weaving_tp(pos_m_path,pos_m_path_end,[a8_wv_distance,Circle_Speed,b1_appro_param,a4_wv_frequency,a3_wv_amplitude,b8_wv_type,wv_direction,current_path,c8_arc_cur_offs],b7_tilt_degree,b3_dealy_all,a9_wv_weldingon,c3_wv_arc,c7_wv_gap,a5_f_hole,b8_wv_2f,a7_weld_crater,squash_l)
          Wait Sleep waitTime=0.5
  Script: write_port_register(weld_done_137,1)
  SuppressedNode
    MoveL speed 400 mm/s, acceleration 800 mm/s^2 (useActiveTCP=true) feature=Base
      MoveDirectionNode (selectedDirection=ZMinus) feature=Joint_6_name
        Until DISTANCE (allowActions=false deceleration=3 distanceNodeType=STOP) Distance=0.03; motionParameters(blendRadius=0)
  wv_direction := 1
  If Auto_W_num[Auto_cur_cell]≥150
    MoveL speed 50 mm/s, acceleration 200 mm/s^2 (useActiveTCP=true) feature=Base
      MoveDirectionNode expression=[-1,1,0.0]
        Until DISTANCE (allowActions=false deceleration=3 distanceNodeType=STOP) Distance=0.03; motionParameters(blendRadius=0)
  ElseIf Auto_W_num[Auto_cur_cell]≥100
    MoveL speed 50 mm/s, acceleration 200 mm/s^2 (useActiveTCP=true) feature=Base
      MoveDirectionNode expression=[-1,-1,0.0]
        Until DISTANCE (allowActions=false deceleration=3 distanceNodeType=STOP) Distance=0.03; motionParameters(blendRadius=0)
  MoveL speed 250 mm/s, acceleration 1200 mm/s^2 (useActiveTCP=true) feature=Base
    MoveDirectionNode (selectedDirection=ZMinus) feature=Joint_6_name
      Until DISTANCE (allowActions=false deceleration=3 distanceNodeType=STOP) Distance=0.03; motionParameters(blendRadius=0)
  Script: homeing()
  If sludge≟1 or (sludge≟2 and current_path>1)
    If not (Auto_W_num[Auto_cur_cell]%10≟1 or Auto_W_num[Auto_cur_cell]%10≟2 or Auto_W_num[Auto_cur_cell]%10≟3)
      pause_trig := True
SubProgram weav_welding_2f (keepSynchronizedWithDisk=false)
  If running_trig≟ True (checkContinuously=true)
    Folder Calculation
      If Auto_W_num[Auto_cur_cell]≟31 or Auto_W_num[Auto_cur_cell]≟32 or Auto_W_num[Auto_cur_cell]≟30
        Folder cal_single
          pos_m_path := A_Touch_p[A_HOR]
          pos_m_path_end := A_Touch_p[A_HOR_R]
          A_middle_weld := interpolate_pose(pos_m_path, pos_m_path_end,0.5)
          Script: A_middle_weld[2]=A_touch_bottom[2]
          A_middle_weld := p[A_middle_weld[0],A_middle_weld[1],A_middle_weld[2],pos_m_path[3],pos_m_path[4],pos_m_path[5]]
      Else 
        SuppressedNode
          side_offset := 10*current_path
        side_offset := 0
        If current_path≟2 or current_path≟4
          SuppressedNode
            center_offset := 15
          center_offset := 0
        Else 
          center_offset := 0
        Folder cal_multi
          pos_m_path := A_Touch_p[A_HOR]
          SuppressedNode
            pos_m_path := pose_trans(pos_m_path, p[side_offset/1000,0,0,0,0,0])
          pos_m_path_end := A_Touch_p[A_HOR_R]
          SuppressedNode
            pos_m_path_end := pose_trans(pos_m_path_end, p[-side_offset/1000,0,0,0,0,0])
          A_middle_weld := interpolate_pose(pos_m_path, pos_m_path_end,0.5)
          Script: A_middle_weld[2]=A_touch_bottom[2]
          SuppressedNode
            A_middle_weld := pose_trans(A_middle_weld, p[-center_offset/1000,0,0,0,0,0])
          A_middle_weld := p[A_middle_weld[0],A_middle_weld[1],A_middle_weld[2],pos_m_path[3],pos_m_path[4],pos_m_path[5]]
      Folder gap_half [hidden by the author, left out]
    Folder Weaving
      If EXT_flag1[6]
        If Auto_W_num[Auto_cur_cell]%10≟1
          Script: inv_inching(inv_inch_time)
          wv_direction := 1
          SuppressedNode
            wv_direction := -1
          step_2f := 1
          Script: welding_result = line_weaving_tp(A_middle_weld,pos_m_path,[a8_wv_distance,Circle_Speed,b1_appro_param,a4_wv_frequency,a3_wv_amplitude,b8_wv_type,wv_direction,current_path,c8_arc_cur_offs],b7_tilt_degree,b3_dealy_all,a9_wv_weldingon,c3_wv_arc,c7_wv_gap,a5_f_hole,b8_wv_2f,a7_weld_crater,squash_l)
          SuppressedNode
            Script: welding_result = line_weaving_tp(pos_m_path,A_middle_weld,[a8_wv_distance,Circle_Speed,b1_appro_param,a4_wv_frequency,a3_wv_amplitude,b8_wv_type,wv_direction,current_path,c8_arc_cur_offs],b7_tilt_degree,b3_dealy_all,a9_wv_weldingon,c3_wv_arc,c7_wv_gap,a5_f_hole,b8_wv_2f,a7_weld_crater,squash_l)
          Wait Sleep waitTime=0.5
        If Auto_W_num[Auto_cur_cell]%10≟2
          Script: inv_inching(inv_inch_time)
          a7_weld_crater := [d_start_current,d_start_voltage,d_start_time,d_end_current_2,d_end_voltage_2,d_end_time_2,d_lean_degree]
          Folder gap_half_right [hidden by the author, left out]
          wv_direction := -1
          SuppressedNode
            wv_direction := 1
          step_2f := 2
          SuppressedNode
            A_middle_weld := feature_offset(A_middle_weld,p[-20/1000,0,0,0,0,0],A_Touch_p[A_sel_v])
          Script: welding_result = line_weaving_tp(A_middle_weld,pos_m_path_end,[a8_wv_distance,Circle_Speed,b1_appro_param,a4_wv_frequency,a3_wv_amplitude,b8_wv_type,wv_direction,current_path,c8_arc_cur_offs],b7_tilt_degree,b3_dealy_all,a9_wv_weldingon,c3_wv_arc,c7_wv_gap,a5_f_hole,b8_wv_2f,a7_weld_crater,squash_l)
          SuppressedNode
            Script: welding_result = line_weaving_tp(pos_m_path_end,A_middle_weld,[a8_wv_distance,Circle_Speed,b1_appro_param,a4_wv_frequency,a3_wv_amplitude,b8_wv_type,wv_direction,current_path,c8_arc_cur_offs],b7_tilt_degree,b3_dealy_all,a9_wv_weldingon,c3_wv_arc,c7_wv_gap,a5_f_hole,b8_wv_2f,a7_weld_crater,squash_l)
      Else 
        If Auto_W_num[Auto_cur_cell]%10≟0
          Script: inv_inching(inv_inch_time)
          wv_direction := 1
          step_2f := 1
          Script: welding_result = line_weaving_tp(pos_m_path,pos_m_path_end,[a8_wv_distance,Circle_Speed,b1_appro_param,a4_wv_frequency,a3_wv_amplitude,b8_wv_type,wv_direction,current_path,c8_arc_cur_offs],b7_tilt_degree,b3_dealy_all,a9_wv_weldingon,c3_wv_arc,c7_wv_gap,a5_f_hole,b8_wv_2f,a7_weld_crater,squash_l)
        Else 
          Script: write_port_register(142,142)
          Halt
  Script: write_port_register(weld_done_137,1)
  MoveL speed 250 mm/s, acceleration 1200 mm/s^2 (useActiveTCP=true) feature=Base
    MoveDirectionNode (selectedDirection=ZMinus) feature=Joint_6_name
      Until DISTANCE (allowActions=false deceleration=3 distanceNodeType=STOP) Distance=0.03; motionParameters(blendRadius=0)
  Script: homeing()
  If sludge≟1 or (sludge≟2 and current_path>1)
    If not (Auto_W_num[Auto_cur_cell]%10≟1)
      pause_trig := True
SubProgram weav_welding_3f [hidden by the author, left out]
SubProgram reset_weld_param [hidden by the author, left out]
